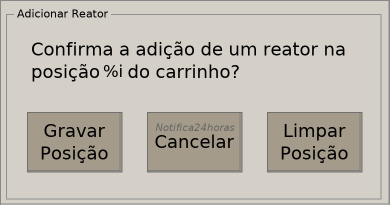
VISUALIZATION ConfigPosicao_Reator_3  // 390x205
VAR_IN_OUT
	bReator: BOOL;
	iOFnumber: INT;
	iSrlNumber: INT;
	
	
	
END_VAR
    GroupBox (6,6 375x193), "Adicionar Reator"
        Label (22,31 332x63), "Confirma a adição de um reator na posição do carrinho?"
        Button (21,106 95x60), "Gravar Posição"
            OnMouseClick: CloseDialog Dialog=ConfigPosicao_Reator_3, Result=OK, NumpadKeypadSet=True
            OnMouseClick: execute { gravarConfigPosicao_Reator_3(); }
        Button (141,106 95x60), "Cancelar"
            OnMouseClick: CloseDialog Dialog=ConfigPosicao_Reator_3, Result=Cancel, NumpadKeypadSet=True
        Rectangle (96,54 22x23), "%i", text variable: GVL.actReat
        Button (261,106 95x60), "Limpar Posição"
            OnMouseClick: CloseDialog Dialog=ConfigPosicao_Reator_3, Result=Cancel, NumpadKeypadSet=True
            OnMouseClick: execute { gvl_p.corPosReator3[gvl.actReat].cor:= 0; }
    Frame (0,0 390x255), invisible if: posCarrinho3.bNotificaTime
        shows Notifica24horas()
END_VISUALIZATION

(* stored: Version 1.1.0.1, ProductVersion 3.1.4024.12
   Visu ConfigPosicao_Reator_3: Id {13583cd1-d758-49be-ac82-e1b8e9591ca1} *)
